INTERFACE I_TestSuite EXTENDS __SYSTEM.IQueryInterface

{attribute 'monitoring' := 'call'}
PROPERTY Duration : LREAL
GET
END_GET
END_PROPERTY

METHOD ReRunIndividualTest
VAR_INPUT
	TestId : T_MaxString;
END_VAR
END_METHOD

METHOD ReRunTests
VAR_INPUT
END_VAR
END_METHOD

METHOD Test : I_TestOperation
VAR_INPUT
	TestId : T_MaxString;
END_VAR
END_METHOD

END_INTERFACE

(* stored: Version 1.1.0.1
   Itf I_TestSuite: Id {d78aa624-4cef-480e-b2e0-77b774c4b77c}
   Property Duration: Id {688b928b-c8ad-4271-8e5d-2d45e72b6796}
   Get Get: Id {625dbe0b-aee5-4131-a28b-442e721555f0}
   Method ReRunIndividualTest: Id {d61aeff6-ac2c-47b8-8bc4-43ae8de6c911}
   Method ReRunTests: Id {cd5b05a7-7512-4eea-b6a2-26305dbec51d}
   Method Test: Id {42521a4e-2eec-4c69-8db8-d94d01afb442} *)
